// TIA Portal V19 export
TYPE "FCP_CONTROL_WORD"
   STRUCT
      Reserved0 : Bool := false;
      Reserved1 : Bool := false;
      Reserved2 : Bool := false;
      Reserved3 : Bool := false;
      Reserved4 : Bool := false;
      Reserved5 : Bool := false;
      Reserved6 : Bool := false;
      Enable : Bool := false;
      Reserved8 : Bool := false;
      Reserved9 : Bool := false;
      Slave : Bool := false;
      ParGroup1 : Bool := false;
      Reserved12 : Bool := false;
      Reserved13 : Bool := false;
      Reserved14 : Bool := false;
      Reserved15 : Bool := false;
   END_STRUCT;
END_TYPE
